FUNCTION_BLOCK DeviceIdentification
VAR
	fb : FB_GetDeviceIdentificationEx;
	initialised : BOOL;
	
	is_windows : BOOL;
	is_windows_ce : BOOL;
	is_bsd : BOOL;
	is_linux : BOOL;
	
	path_delimiter : STRING(1);
END_VAR

METHOD PUBLIC Initialise : BOOL
VAR
	dev_id : Tc2_Utilities.ST_DeviceIdentificationEx;
END_VAR
IF initialised THEN
	Initialise := initialised;
	RETURN;
END_IF

fb(bExecute := TRUE);

IF NOT fb.bBusy THEN
	dev_id := fb.stDevIdent;
	initialised := TRUE;
	fb(bExecute := FALSE);
END_IF

IF Left(dev_id.strImageOsName, 10) = 'Windows CE' THEN
	is_windows_ce := TRUE;
ELSIF Left(dev_id.strImageOsName, 7) = 'Windows' THEN
	is_windows := TRUE; 
END_IF

IF is_windows OR is_windows_ce THEN
	path_delimiter := '\';
ELSE
	path_delimiter := '/';
END_IF
END_METHOD

{attribute 'monitoring':='call'}
PROPERTY PUBLIC IsBsd : BOOL
GET // PUBLIC
IsBsd := is_bsd;
END_GET
END_PROPERTY

{attribute 'monitoring':='call'}
PROPERTY PUBLIC IsLinux : BOOL
GET // PUBLIC
IsLinux := is_linux;
END_GET
END_PROPERTY

{attribute 'monitoring':='call'}
PROPERTY PUBLIC IsWindows : BOOL
GET // PUBLIC
IsWindows := is_windows;
END_GET
END_PROPERTY

{attribute 'monitoring':='call'}
PROPERTY PUBLIC IsWindowsCE : BOOL
GET // PUBLIC
IsWindowsCE := is_windows_ce;
END_GET
END_PROPERTY

{attribute 'monitoring':='call'}
PROPERTY PUBLIC PathDelimiter : STRING(1)
GET // PUBLIC
PathDelimiter := path_delimiter;
END_GET
END_PROPERTY

END_FUNCTION_BLOCK

(* stored: Version 1.1.0.1
   POU DeviceIdentification: Id {41fc405e-dc1d-4522-98e4-8d210b8f7d50}, SpecialFunc None
   Method Initialise: Id {cd70b8ec-64d4-4b8d-b42f-1333153b7073}
   Property IsBsd: Id {09f6f01d-7068-4c14-a3e9-1e8c3477e6fb}
   Get Get: Id {7b10fac7-b026-4d23-9c77-11934fe53f48}
   Property IsLinux: Id {225311cc-30d5-431c-b75d-2b9479e339ea}
   Get Get: Id {67bbca29-c393-4c21-9195-8a0eb4c78ba2}
   Property IsWindows: Id {f5f78fb3-64e0-4d0e-a69f-ed0311e82b82}
   Get Get: Id {f7959264-2227-4e17-b992-7bddf0a7de28}
   Property IsWindowsCE: Id {447f6a2a-6d07-4b1d-b45f-926eb9f4c9bd}
   Get Get: Id {c56364d1-6325-4283-bcf3-adbfca7e0cba}
   Property PathDelimiter: Id {9908fc20-c991-4bd4-8ef7-825bd3e51254}
   Get Get: Id {9108cfab-a7b2-4ee6-9f74-96c0172d3875} *)
